{attribute 'GeneratedUsingTerminal: KL2300-0100'}
{attribute addProperty BoxType "KL2300-0100"}
{attribute addProperty Id "InputAT %I*BOOL0OutputAT %Q*BOOL0"}
{attribute addProperty CRC "1892259827"}
{attribute addProperty Size "0"}
TYPE Channel_70C997F3 :
STRUCT
	{attribute addProperty Name "Input"}
	Input AT %I* : BOOL;
	{attribute addProperty Name "Output"}
	Output AT %Q* : BOOL;
END_STRUCT
END_TYPE

(* stored: Version 1.2.0.0, ProductVersion 3.1.4024.9
   DUT Channel_70C997F3: Id {9659ddbf-ced7-46cc-b885-493107389f23} *)
